Staubli VAL3: newMoveCmd.pjx

Parameters version=s7.9.1 stackSize=5000 millimeterUnit=true
Program file=newMoveCmd.pgx
Program file=start.pgx
Program file=stop.pgx
Data file=newMoveCmd.dtx
Type name=CartesianSpace path=Disk://RobotController_Libs/RobotStatus/CartesianSpace/CartesianSpace.pjx
Type name=ModelParameter path=Disk://RobotController_Libs/ModelParameter/ModelParameter.pjx
Type name=JointSpace path=Disk://RobotController_Libs/RobotStatus/JointSpace/JointSpace.pjx
Type name=RobotCfgStatus path=Disk://RobotController_Libs/RobotCfgStatus/RobotCfgStatus.pjx
